// TIA Portal V17 export
// export: Created 2025-01-08T13:55:37.6994246Z, ExportSetting WithDefaults, DisplayName Totally Integrated Automation Portal, DisplayVersion V17, DisplayName TIA Portal Openness, DisplayVersion V17, DisplayName TIA Portal Version Control Interface, DisplayVersion V17, DisplayName SINAMICS Startdrive Advanced, DisplayVersion V17 Update2, DisplayName SINAMICS Startdrive G130, G150, S120, S150, SINAMICS MV, S210, DisplayVersion V17 Update2, DisplayName SINAMICS Startdrive G110M, G120, G120C, G120D, G120P, G115D, DisplayVersion V17 Update2, DisplayName STEP 7 Professional, DisplayVersion V17, DisplayName STEP 7 Safety, DisplayVersion V17, DisplayName WinCC Advanced, DisplayVersion V17
TYPE "HSMMachineParaMask8"
// stored: IsFailsafeCompliant false
   STRUCT
      MPARA_I_Reserve_42 : Bool;
      MPARA_I_Reserve_43 : Bool;
      MPARA_I_Reserve_44 : Bool;
      MPARA_I_Reserve_45 : Bool;
      MPARA_I_Reserve_46 : Bool;
      MPARA_I_Reserve_47 : Bool;
      MPARA_I_Reserve_48 : Bool;
      MPARA_I_Reserve_49 : Bool;
      MPARA_I_Reserve_50 : Bool;
      MPARA_I_Reserve_51 : Bool;
      MPARA_I_Reserve_52 : Bool;
      MPARA_I_Reserve_53 : Bool;
      MPARA_I_Reserve_54 : Bool;
      MPARA_I_Reserve_55 : Bool;
      MPARA_I_Reserve_56 : Bool;
      MPARA_I_Reserve_57 : Bool;
   END_STRUCT;
END_TYPE
